PROGRAM MAIN
VAR
	XMLTesten : XMLTesten;
END_VAR

XMLTesten();

END_PROGRAM

(* stored: Version 1.1.0.1, ProductVersion 3.1.4024.3
   POU MAIN: Id {ea0b4a2c-0bed-406f-a5c3-9ef6d33ee418}, SpecialFunc None *)
